TYPE ST_SequenceIn :
STRUCT
END_STRUCT
END_TYPE

(* stored: Version 1.1.0.1
   DUT ST_SequenceIn: Id {891c0004-6029-091d-0228-3887352079f1} *)
